PROGRAM PRG_Reference_POU
VAR
	
	fbTimersTEST	: FB_TimersTEST;
	
	tTON_Q			: BOOL;
	tTOF_Q			: BOOL;
	
	tTimer			: TIME := T#4S;
	
	bStartTON		: BOOL;
	bStartTOF		: BOOL;
	
	
END_VAR


fbTimersTEST(
	bStartTON:= bStartTON, 
	bStartTOF:= bStartTOF, 
	tTime:= tTimer, 
	tTON:= GVL_test.stFBinside.aTONs[1],
	tTOF:= GVL_test.stFBinside.aTOFs[1],
	tTON_Q=> tTON_Q, 
	tTOF_Q=> tTOF_Q
);

END_PROGRAM

(* stored: Version 1.1.0.1
   POU PRG_Reference_POU: Id {79c550d0-418d-4bc2-9d62-dc1d499218cc}, SpecialFunc None *)
